// TIA Portal V20 export
DATA_BLOCK "InstCounterDataset2"   // DB66
TITLE = Instance CounterDataSet2
{ DB_Accessible_From_OPC_UA := 'FALSE' }
AUTHOR : SICAR
FAMILY : ProdData
// Instance DB
// stored: DBAccessibleFromOPCUA false, InstanceOfName LSicar_ProdDataCounter, InstanceOfType FB
"LSicar_ProdDataCounter"
   // VAR_INPUT
   //    numberConfigDataSets { ExternalAccessible := 'False'; ExternalVisible := 'False'; ExternalWritable := 'False'} : Int;
   //    dataSetNumber { ExternalAccessible := 'False'; ExternalVisible := 'False'; ExternalWritable := 'False'} : UInt;
   // END_VAR
   // VAR_IN_OUT
   //    numberOfDataSets : "LSicar_typeNumberOfDataSets";
   //    dataSet : "LSicar_typeCounter";
   // END_VAR
   // VAR
   //    statCounter { ExternalAccessible := 'False'; ExternalVisible := 'False'; ExternalWritable := 'False'} : Array[0..20] of "LSicar_typeEdgePulseStruct";
   //    statRisEdgeResetAllExt { ExternalAccessible := 'False'; ExternalVisible := 'False'; ExternalWritable := 'False'} : Bool;
   //    statPosPulseResetAllExt { ExternalAccessible := 'False'; ExternalVisible := 'False'; ExternalWritable := 'False'} : Bool;
   //    statRisEdgeResetAll { ExternalAccessible := 'False'; ExternalVisible := 'False'; ExternalWritable := 'False'} : Bool;
   //    statPosPulseResetAll { ExternalAccessible := 'False'; ExternalVisible := 'False'; ExternalWritable := 'False'} : Bool;
   // END_VAR
BEGIN
END_DATA_BLOCK
